FUNCTION_BLOCK SET_AT_INDEX (* Set value of array at given index. Data types of value to be set must correspond to the array data type. Data type of resulting output array must correspond to input array data type. *)
  (* Description: Copyright (c) 2014 Profactor GmbH This program and the accompanying materials are made available under the terms of the Eclipse Public License 2.0 which is available at https://www.eclipse.org/legal/epl-2.0/ SPDX-License-Identifier: EPL-2.0 *)
  (* Version 1.0, 2014-08-05, Matthias Plasch, Profactor GmbH *)
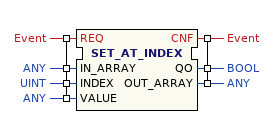
  EVENT_INPUT
    REQ WITH IN_ARRAY, INDEX, VALUE; (* Service Request *)
  END_EVENT
  EVENT_OUTPUT
    CNF WITH QO, OUT_ARRAY; (* Confirmation of Requested Service *)
  END_EVENT
  VAR_INPUT
    IN_ARRAY : ANY; (* input array *)
    INDEX : UINT; (* index to fetch value from *)
    VALUE : ANY; (* value to be copied to given index *)
  END_VAR
  VAR_OUTPUT
    QO : BOOL; (* Event Output Qualifier *)
    OUT_ARRAY : ANY; (* resulting array after set *)
  END_VAR
END_FUNCTION_BLOCK
